FUNCTION_BLOCK PUBLIC FB_Conv3
VAR_INPUT
	Conv4_IsOpen		:	BOOL	;
END_VAR
VAR_OUTPUT	
END_VAR
VAR
	
	Set_Motor	:	BOOL		;
	Reset_Motor	:	BOOL		;
	iSTEP		:	INT := 0	;
	Timer1		:	TON			;
	Timer2		:	TON			;
	Timer3		:	TON			;

END_VAR

CASE iSTEP OF 

	// ================================================ conv3 motor init	
	(*conv motor intialization*)
	0:	IF IO.bConv_Ready AND IO_control.bEstop THEN
			IO_control.bMotor3 := FALSE;
			iSTEP := iSTEP + 1 ;
		END_IF
	
	// ================================================ check for open status for next conv
	1:	IF IO_Conveyor.bExit3_IsOpen THEN		
			iSTEP := iSTEP + 1 	;
		END_IF
	
	// ================================================ motor2 n motor3 to start when conv2 out is ON	
	2:	IF IO_Conveyor.Conv2_Done THEN
			IO_control.bMotor2 S= IO_Conveyor.Conv2_Done ;
			IO_control.bMotor3 S= IO_Conveyor.Conv2_Done ;
			iSTEP := iSTEP + 1 ;
		END_IF
	
	// ================================================ motor2 to stop if bconv3 in is ON		
	3:	IF IO.bConv3_In THEN
			IO_control.bMotor2 R= IO.bConv3_In ;
			IO_Conveyor.Conv2_Done := FALSE ;
			iSTEP := iSTEP + 1 ;
		END_IF
	
	// ================================================ stop motor3 if conv3_out ON	
	4:	IF IO.bConv3_Out THEN
			IO_control.bMotor3 R= IO.bConv3_Out ;
			IO_Conveyor.Conv3_Done := TRUE;
			iSTEP := iSTEP + 1;
		END_IF

	// ================================================ receive feedback from conv4	
	5:	IF NOT IO_Conveyor.Conv3_Done THEN
			iSTEP := 0 ;
		END_IF
		
END_CASE

IF IO_control.bReset AND IO.bManualMode THEN
	IO_Conveyor.Conv3_Done := FALSE;
	iSTEP := 0 ;
END_IF

END_FUNCTION_BLOCK

(* stored: Version 1.1.0.1, ProductVersion 3.1.4024.12
   POU FB_Conv3: Id {0ccdce00-e922-4b28-aa2f-495500201879}, SpecialFunc None *)
